(* IEC 61131-3 sources: wafer-proc-sim/plc, 4 files *)

(* ---- InterlockFB.st ---- *)
(*
 * InterlockFB.st — Safety interlock monitor Function Block
 * IEC 61131-3 Structured Text  /  IEC 61508 SIL-1 inspired
 *
 * Each sensor has WARN / STOP / FAULT thresholds.
 * FAULT latches E_STOP until operator reset.
 *)

FUNCTION_BLOCK InterlockFB
VAR_INPUT
    Spindle_rpm     : REAL;     (* spindle speed readback *)
    Coolant_lpm     : REAL;     (* coolant flow [L/min] *)
    Door_closed     : BOOL;     (* safety door sensor *)
    BladeDepth_mm   : REAL;     (* blade Z position [mm, negative = into wafer] *)
    ChuckVac_kPa    : REAL;     (* chuck vacuum [kPa] *)
    BladeWear_um    : REAL;     (* estimated blade wear [µm] *)
    Reset           : BOOL;     (* operator reset pulse *)
END_VAR

VAR_OUTPUT
    System_OK       : BOOL;     (* TRUE = safe to run *)
    E_Stop          : BOOL;     (* latched emergency stop *)
    WarnActive      : BOOL;     (* at least one WARN *)
    FaultCode       : INT;      (* 0=OK 1=SpindleOvspd 2=NoCoolant
                                   3=DoorOpen 4=BladeDeep 5=VacLow
                                   6=WearHigh *)
END_VAR

VAR
    (* threshold constants *)
    SP_WARN_HI  : REAL := 32000.0;
    SP_FAULT_HI : REAL := 35000.0;
    CL_FAULT_LO : REAL := 0.5;
    BD_WARN_LO  : REAL := -0.35;
    BD_FAULT_LO : REAL := -0.50;
    VC_WARN_LO  : REAL := 60.0;
    WR_WARN_HI  : REAL := 30.0;
    WR_FAULT_HI : REAL := 50.0;

    _estop_latch : BOOL := FALSE;
END_VAR

    (* Reset latch on rising edge of Reset *)
    IF Reset AND _estop_latch THEN
        _estop_latch := FALSE;
    END_IF

    WarnActive := FALSE;
    FaultCode  := 0;

    (* Check spindle overspeed *)
    IF ABS(Spindle_rpm) > SP_FAULT_HI THEN
        _estop_latch := TRUE;
        FaultCode    := 1;
    ELSIF ABS(Spindle_rpm) > SP_WARN_HI THEN
        WarnActive := TRUE;
    END_IF

    (* Check coolant flow *)
    IF Coolant_lpm < CL_FAULT_LO THEN
        _estop_latch := TRUE;
        IF FaultCode = 0 THEN FaultCode := 2; END_IF
    END_IF

    (* Check door *)
    IF NOT Door_closed THEN
        _estop_latch := TRUE;
        IF FaultCode = 0 THEN FaultCode := 3; END_IF
    END_IF

    (* Check blade depth (more negative = deeper cut) *)
    IF BladeDepth_mm < BD_FAULT_LO THEN
        _estop_latch := TRUE;
        IF FaultCode = 0 THEN FaultCode := 4; END_IF
    ELSIF BladeDepth_mm < BD_WARN_LO THEN
        WarnActive := TRUE;
    END_IF

    (* Check chuck vacuum *)
    IF ChuckVac_kPa < VC_WARN_LO THEN
        WarnActive := TRUE;
        IF FaultCode = 0 THEN FaultCode := 5; END_IF
    END_IF

    (* Check blade wear *)
    IF BladeWear_um > WR_FAULT_HI THEN
        _estop_latch := TRUE;
        IF FaultCode = 0 THEN FaultCode := 6; END_IF
    ELSIF BladeWear_um > WR_WARN_HI THEN
        WarnActive := TRUE;
    END_IF

    E_Stop    := _estop_latch;
    System_OK := NOT _estop_latch;

END_FUNCTION_BLOCK

(* ---- RecipeSeqFB.st ---- *)
(*
 * RecipeSeqFB.st — Dicing recipe sequencer Function Block
 * IEC 61131-3 Structured Text
 *
 * Drives the 12-step DISCO dicing recipe as a CASE state machine.
 * Interlocks are checked at every scan.
 *)

FUNCTION_BLOCK RecipeSeqFB
VAR_INPUT
    Start       : BOOL;     (* operator start command *)
    Abort       : BOOL;     (* operator abort *)
    StepDone    : BOOL;     (* rising edge = current step completed *)
    Interlock_OK: BOOL;     (* from InterlockFB.System_OK *)
    dt_ms       : REAL := 1.0;
END_VAR

VAR_OUTPUT
    State       : INT;      (* 0=IDLE 1=RUNNING 2=DONE 3=FAULT *)
    StepIndex   : INT;      (* 0..11 *)
    StepName    : STRING;
    Progress_pct: REAL;
    Fault       : BOOL;
END_VAR

VAR
    _elapsed_ms     : REAL := 0.0;
    _step_done_prev : BOOL := FALSE;
    _step_done_rise : BOOL;

    (* Step timeouts [ms] *)
    TIMEOUT : ARRAY[0..11] OF REAL := [
        5000.0,   (* 0  LOAD_WAFER     *)
        2000.0,   (* 1  VACUUM_ON      *)
        8000.0,   (* 2  ALIGN_WAFER    *)
        3000.0,   (* 3  PRIME_SPINDLE  *)
        1000.0,   (* 4  COOLANT_ON     *)
        60000.0,  (* 5  CUT_X_STREETS  *)
        2000.0,   (* 6  ROTATE_CHUCK   *)
        60000.0,  (* 7  CUT_Y_STREETS  *)
        2000.0,   (* 8  RETRACT_BLADE  *)
        1000.0,   (* 9  COOLANT_OFF    *)
        3000.0,   (* 10 SPINDLE_OFF    *)
        5000.0    (* 11 UNLOAD_WAFER   *)
    ];

    STEP_NAMES : ARRAY[0..11] OF STRING := [
        'LOAD_WAFER', 'VACUUM_ON', 'ALIGN_WAFER', 'PRIME_SPINDLE',
        'COOLANT_ON', 'CUT_X_STREETS', 'ROTATE_CHUCK', 'CUT_Y_STREETS',
        'RETRACT_BLADE', 'COOLANT_OFF', 'SPINDLE_OFF', 'UNLOAD_WAFER'
    ];

    TOTAL_STEPS : INT := 12;
END_VAR

    (* Detect rising edge on StepDone *)
    _step_done_rise := StepDone AND NOT _step_done_prev;
    _step_done_prev := StepDone;

    CASE State OF

        0: (* IDLE *)
            StepIndex   := 0;
            Progress_pct := 0.0;
            _elapsed_ms  := 0.0;
            Fault        := FALSE;
            IF Start AND Interlock_OK THEN
                State := 1;
            END_IF

        1: (* RUNNING *)
            StepName := STEP_NAMES[StepIndex];
            Progress_pct := REAL_TO_REAL(StepIndex) / REAL_TO_REAL(TOTAL_STEPS) * 100.0;

            IF NOT Interlock_OK OR Abort THEN
                State := 3;  (* → FAULT *)
            END_IF

            _elapsed_ms := _elapsed_ms + dt_ms;

            (* Timeout check *)
            IF _elapsed_ms > TIMEOUT[StepIndex] THEN
                State := 3;
                Fault := TRUE;
            END_IF

            (* Step complete *)
            IF _step_done_rise THEN
                _elapsed_ms := 0.0;
                IF StepIndex >= TOTAL_STEPS - 1 THEN
                    State        := 2;
                    Progress_pct := 100.0;
                ELSE
                    StepIndex := StepIndex + 1;
                END_IF
            END_IF

        2: (* DONE *)
            Fault := FALSE;

        3: (* FAULT *)
            Fault := TRUE;
            IF NOT Abort AND Start AND Interlock_OK THEN
                State     := 0;  (* reset to IDLE after operator clears *)
                StepIndex := 0;
            END_IF

    END_CASE

END_FUNCTION_BLOCK

(* ---- SpindleFB.st ---- *)
(*
 * SpindleFB.st — PMSM spindle Function Block
 * IEC 61131-3 Structured Text
 *
 * Models the dq-axis dynamics of the DISCO dicing saw spindle motor.
 * Called every control cycle (dt_us = 10 µs).
 *)

FUNCTION_BLOCK SpindleFB
VAR_INPUT
    Enable      : BOOL;         (* TRUE = run spindle *)
    SpeedRef_rpm: REAL;         (* target speed [rpm] *)
    dt_us       : REAL := 10.0; (* timestep [µs] *)
END_VAR

VAR_OUTPUT
    Speed_rpm   : REAL;         (* actual speed [rpm] *)
    Torque_Nm   : REAL;         (* electromagnetic torque *)
    I_q         : REAL;         (* q-axis current [A] *)
    I_d         : REAL;         (* d-axis current [A] *)
    Fault       : BOOL;         (* overspeed / overcurrent *)
END_VAR

VAR
    (* Motor params — DISCO high-speed spindle *)
    Rs          : REAL := 0.5;      (* stator resistance [Ω] *)
    Ld          : REAL := 0.0015;   (* d-axis inductance [H] *)
    Lq          : REAL := 0.0015;   (* q-axis inductance [H] *)
    Psi_f       : REAL := 0.08;     (* flux linkage [Wb] *)
    Pn          : REAL := 4.0;      (* pole pairs *)
    J           : REAL := 0.0001;   (* rotor inertia [kg·m²] *)
    B_fric      : REAL := 0.01;     (* viscous friction [N·m·s] *)

    (* PI current controller *)
    Kp_i        : REAL := 10.0;
    Ki_i        : REAL := 50.0;
    Iq_ref      : REAL;
    Err_q       : REAL;
    Int_iq      : REAL := 0.0;
    V_d         : REAL;
    V_q         : REAL;

    (* State *)
    Omega_rad_s : REAL := 0.0;  (* mechanical angular velocity [rad/s] *)
    _I_d        : REAL := 0.0;
    _I_q        : REAL := 0.0;
    dt_s        : REAL;

    (* Limits *)
    MAX_SPEED_RPM  : REAL := 35000.0;
    MAX_CURRENT_A  : REAL := 25.0;
END_VAR

    IF NOT Enable THEN
        Omega_rad_s := Omega_rad_s * 0.99;  (* coast-down *)
        Speed_rpm   := Omega_rad_s * 60.0 / (2.0 * 3.14159);
        Fault       := FALSE;
        RETURN;
    END_IF

    dt_s := dt_us * 1.0E-6;

    (* Speed controller → Iq reference *)
    Iq_ref := (SpeedRef_rpm * 2.0 * 3.14159 / 60.0 - Omega_rad_s) * 5.0;
    Iq_ref := LIMIT(-20.0, Iq_ref, 20.0);

    (* PI current controller (q-axis) *)
    Err_q  := Iq_ref - _I_q;
    Int_iq := Int_iq + Err_q * dt_s;
    V_q    := Kp_i * Err_q + Ki_i * Int_iq
              + Pn * Omega_rad_s * (Ld * _I_d + Psi_f);   (* feed-forward *)
    V_d    := Kp_i * (0.0 - _I_d)
              - Pn * Omega_rad_s * Lq * _I_q;

    (* dq current integration *)
    _I_d := _I_d + (V_d - Rs * _I_d + Pn * Omega_rad_s * Lq * _I_q) / Ld * dt_s;
    _I_q := _I_q + (V_q - Rs * _I_q - Pn * Omega_rad_s * (Ld * _I_d + Psi_f)) / Lq * dt_s;

    (* Mechanical dynamics *)
    Torque_Nm   := 1.5 * Pn * (Psi_f * _I_q + (Ld - Lq) * _I_d * _I_q);
    Omega_rad_s := Omega_rad_s + (Torque_Nm - B_fric * Omega_rad_s) / J * dt_s;

    (* Outputs *)
    Speed_rpm := Omega_rad_s * 60.0 / (2.0 * 3.14159);
    I_q       := _I_q;
    I_d       := _I_d;

    (* Fault detection *)
    Fault := (ABS(Speed_rpm) > MAX_SPEED_RPM) OR (ABS(_I_q) > MAX_CURRENT_A);

END_FUNCTION_BLOCK

(* ---- DicingController.st ---- *)
(*
 * DicingController.st — Top-level DISCO dicing saw PLC program
 * IEC 61131-3 Structured Text
 *
 * Integrates SpindleFB, InterlockFB, RecipeSeqFB into one scan cycle.
 * Mirrors the real machine controller architecture: each FB encapsulates
 * one subsystem; the main PROGRAM wires I/O and coordinates state.
 *
 * Compile with: OpenPLC Runtime  or  CODESYS V3.5
 *)

PROGRAM DicingController

VAR
    (* Function block instances *)
    Spindle     : SpindleFB;
    Interlock   : InterlockFB;
    Recipe      : RecipeSeqFB;

    (* HMI inputs (written by operator panel / SCADA) *)
    HMI_Start       : BOOL := FALSE;
    HMI_Abort       : BOOL := FALSE;
    HMI_Reset       : BOOL := FALSE;
    HMI_SpeedRef    : REAL := 30000.0;  (* [rpm] *)

    (* Sensor inputs (mapped to physical I/O in real machine) *)
    IN_CoolantFlow  : REAL := 2.0;      (* [L/min] *)
    IN_DoorClosed   : BOOL := TRUE;
    IN_BladeDepth   : REAL := 0.0;      (* [mm] *)
    IN_ChuckVac     : REAL := 80.0;     (* [kPa] *)
    IN_BladeWear    : REAL := 0.0;      (* [µm] — from APC/EnKF *)

    (* Internal *)
    StepDone_pulse  : BOOL := FALSE;
    dt_ms           : REAL := 1.0;      (* scan cycle [ms] *)

    (* Status outputs (to HMI / data logger) *)
    OUT_Speed_rpm   : REAL;
    OUT_Torque_Nm   : REAL;
    OUT_RecipeState : INT;
    OUT_StepName    : STRING;
    OUT_Progress    : REAL;
    OUT_EStop       : BOOL;
    OUT_FaultCode   : INT;
END_VAR

    (* 1. Interlock evaluation — always first *)
    Interlock(
        Spindle_rpm   := OUT_Speed_rpm,
        Coolant_lpm   := IN_CoolantFlow,
        Door_closed   := IN_DoorClosed,
        BladeDepth_mm := IN_BladeDepth,
        ChuckVac_kPa  := IN_ChuckVac,
        BladeWear_um  := IN_BladeWear,
        Reset         := HMI_Reset
    );

    (* 2. Recipe sequencer *)
    Recipe(
        Start        := HMI_Start,
        Abort        := HMI_Abort OR Interlock.E_Stop,
        StepDone     := StepDone_pulse,
        Interlock_OK := Interlock.System_OK,
        dt_ms        := dt_ms
    );

    (* 3. Spindle — only run when recipe is active and interlocks clear *)
    Spindle(
        Enable       := Interlock.System_OK AND (Recipe.State = 1),
        SpeedRef_rpm := HMI_SpeedRef,
        dt_us        := 10.0
    );

    (* 4. Propagate fault from spindle back to interlock *)
    IF Spindle.Fault THEN
        HMI_Abort := TRUE;
    END_IF

    (* 5. Collect outputs for HMI *)
    OUT_Speed_rpm   := Spindle.Speed_rpm;
    OUT_Torque_Nm   := Spindle.Torque_Nm;
    OUT_RecipeState := Recipe.State;
    OUT_StepName    := Recipe.StepName;
    OUT_Progress    := Recipe.Progress_pct;
    OUT_EStop       := Interlock.E_Stop;
    OUT_FaultCode   := Interlock.FaultCode;

END_PROGRAM
